// TwinCAT 3 PLC project HardwareSimulator
// ProgramVersion: 3.1.4024.0
// libraries:
//   Tc2_Standard, * (Beckhoff Automation GmbH)
//   Tc2_System, * (Beckhoff Automation GmbH)
//   Tc2_Utilities, * (Beckhoff Automation GmbH)
//   Tc3_Module, * (Beckhoff Automation GmbH)
//   VisuSymbols,3.5.10.0,System
// project tree:
//   / GlobalTextList.TcGTLO (not stored), PlcTask.TcTTO (not stored), Visualization Manager.TcVMO (not stored)
//   POUs/ MAIN.TcPOU, SIM_ValveWithFB.TcPOU, SIM_ValveWithDoubleFB.TcPOU, SIM_MOVITRAC_B.TcPOU (not stored)
//   VISUs/ Visualization.TcVIS (not stored)
// (motion and I/O tree: see PLC project cleanroomconnect)
// real-time tasks:
//   TASK PlcTask: cycle T#10ms, priority 20, ADS port 350
//   TASK PlcTask1: cycle T#10ms, priority 21, ADS port 351
//   TASK VISU_TASK: cycle T#200000us, priority 30, ADS port 352
// variable links:
//   CleanroomConnect/CleanroomConnect Instance <-> HardwareSimulator/HardwareSimulator Instance
//     PlcTask Inputs/GVL_Modules.g_emDockingInterface.s_cmDockingClampsLower.I_bStaValveIsOff <-> PlcTask Outputs/MAIN.simDockingClampLower.Q_bStaFeedbackOff
//     PlcTask Inputs/GVL_Modules.g_emDockingInterface.s_cmDockingClampsLower.I_bStaValveIsOff2 <-> PlcTask Outputs/MAIN.simDockingClampLower.Q_bStaFeedbackOff2
//     PlcTask Inputs/GVL_Modules.g_emDockingInterface.s_cmDockingClampsLower.I_bStaValveIsOn <-> PlcTask Outputs/MAIN.simDockingClampLower.Q_bStaFeedbackOn
//     PlcTask Inputs/GVL_Modules.g_emDockingInterface.s_cmDockingClampsLower.I_bStaValveIsOn2 <-> PlcTask Outputs/MAIN.simDockingClampLower.Q_bStaFeedbackOn2
//     PlcTask Inputs/GVL_Modules.g_emDockingInterface.s_cmDockingClampsUpper.I_bStaValveIsOff <-> PlcTask Outputs/MAIN.simDockingClampUpper.Q_bStaFeedbackOff
//     PlcTask Inputs/GVL_Modules.g_emDockingInterface.s_cmDockingClampsUpper.I_bStaValveIsOff2 <-> PlcTask Outputs/MAIN.simDockingClampUpper.Q_bStaFeedbackOff2
//     PlcTask Inputs/GVL_Modules.g_emDockingInterface.s_cmDockingClampsUpper.I_bStaValveIsOn <-> PlcTask Outputs/MAIN.simDockingClampUpper.Q_bStaFeedbackOn
//     PlcTask Inputs/GVL_Modules.g_emDockingInterface.s_cmDockingClampsUpper.I_bStaValveIsOn2 <-> PlcTask Outputs/MAIN.simDockingClampUpper.Q_bStaFeedbackOn2
//     PlcTask Inputs/GVL_Modules.g_emDockingInterface.s_cmDoorOpener.I_bStaValveIsOff <-> PlcTask Outputs/MAIN.simDoorOpener.Q_bStaFeedbackOff
//     PlcTask Inputs/GVL_Modules.g_emDockingInterface.s_cmDoorOpener.I_bStaValveIsOn <-> PlcTask Outputs/MAIN.simDoorOpener.Q_bStaFeedbackOn
//     PlcTask Inputs/GVL_Modules.g_emDockingInterface.s_cmDoorShutter.I_bStaValveIsOff <-> PlcTask Outputs/MAIN.simDoorShutter.Q_bStaFeedbackOff
//     PlcTask Inputs/GVL_Modules.g_emDockingInterface.s_cmDoorShutter.I_bStaValveIsOn <-> PlcTask Outputs/MAIN.simDoorShutter.Q_bStaFeedbackOn
//     PlcTask Inputs/GVL_Modules.g_emDockingInterface.s_cmUnlockingPinLower.I_bStaValveIsOff <-> PlcTask Outputs/MAIN.simUnlockPinLower.Q_bStaFeedbackOff
//     PlcTask Inputs/GVL_Modules.g_emDockingInterface.s_cmUnlockingPinLower.I_bStaValveIsOn <-> PlcTask Outputs/MAIN.simUnlockPinLower.Q_bStaFeedbackOn
//     PlcTask Inputs/GVL_Modules.g_emDockingInterface.s_cmUnlockingPinUpper.I_bStaValveIsOff <-> PlcTask Outputs/MAIN.simUnlockPinUpper.Q_bStaFeedbackOff
//     PlcTask Inputs/GVL_Modules.g_emDockingInterface.s_cmUnlockingPinUpper.I_bStaValveIsOn <-> PlcTask Outputs/MAIN.simUnlockPinUpper.Q_bStaFeedbackOn
//     PlcTask Inputs/GVL_Modules.g_emPalletConveyor.s_cmCentringUnit.I_bStaValveIsOff <-> PlcTask Outputs/MAIN.simCentring.Q_bStaFeedbackOff
//     PlcTask Inputs/GVL_Modules.g_emPalletConveyor.s_cmCentringUnit.I_bStaValveIsOff2 <-> PlcTask Outputs/MAIN.simCentring.Q_bStaFeedbackOff2
//     PlcTask Inputs/GVL_Modules.g_emPalletConveyor.s_cmCentringUnit.I_bStaValveIsOn <-> PlcTask Outputs/MAIN.simCentring.Q_bStaFeedbackOn
//     PlcTask Inputs/GVL_Modules.g_emPalletConveyor.s_cmCentringUnit.I_bStaValveIsOn2 <-> PlcTask Outputs/MAIN.simCentring.Q_bStaFeedbackOn2
//     PlcTask Inputs/GVL_Modules.g_emPalletConveyor.s_cmPalletConveyor.I_bStaMotorIsRunning <-> PlcTask Outputs/MAIN.sim_MOVITRAC_B.Q_bStaMotorIsRunning
//     PlcTask Inputs/GVL_Modules.g_emPalletConveyor.s_cmPalletConveyor.I_bStaReadyForOperation <-> PlcTask Outputs/MAIN.sim_MOVITRAC_B.Q_bStaReadyForOperation
//     PlcTask Outputs/GVL_Modules.g_emDockingInterface.s_cmDockingClampsLower.Q_bCmdOff <-> PlcTask Inputs/MAIN.simDockingClampLower.I_bCmdValveOff
//     PlcTask Outputs/GVL_Modules.g_emDockingInterface.s_cmDockingClampsLower.Q_bCmdOn <-> PlcTask Inputs/MAIN.simDockingClampLower.I_bCmdValveOn
//     PlcTask Outputs/GVL_Modules.g_emDockingInterface.s_cmDockingClampsUpper.Q_bCmdOff <-> PlcTask Inputs/MAIN.simDockingClampUpper.I_bCmdValveOff
//     PlcTask Outputs/GVL_Modules.g_emDockingInterface.s_cmDockingClampsUpper.Q_bCmdOn <-> PlcTask Inputs/MAIN.simDockingClampUpper.I_bCmdValveOn
//     PlcTask Outputs/GVL_Modules.g_emDockingInterface.s_cmDoorOpener.Q_bCmdOff <-> PlcTask Inputs/MAIN.simDoorOpener.I_bCmdValveOff
//     PlcTask Outputs/GVL_Modules.g_emDockingInterface.s_cmDoorOpener.Q_bCmdOn <-> PlcTask Inputs/MAIN.simDoorOpener.I_bCmdValveOn
//     PlcTask Outputs/GVL_Modules.g_emDockingInterface.s_cmDoorShutter.Q_bCmdOff <-> PlcTask Inputs/MAIN.simDoorShutter.I_bCmdValveOff
//     PlcTask Outputs/GVL_Modules.g_emDockingInterface.s_cmDoorShutter.Q_bCmdOn <-> PlcTask Inputs/MAIN.simDoorShutter.I_bCmdValveOn
//     PlcTask Outputs/GVL_Modules.g_emDockingInterface.s_cmUnlockingPinLower.Q_bCmdOff <-> PlcTask Inputs/MAIN.simUnlockPinLower.I_bCmdValveOff
//     PlcTask Outputs/GVL_Modules.g_emDockingInterface.s_cmUnlockingPinLower.Q_bCmdOn <-> PlcTask Inputs/MAIN.simUnlockPinLower.I_bCmdValveOn
//     PlcTask Outputs/GVL_Modules.g_emDockingInterface.s_cmUnlockingPinUpper.Q_bCmdOff <-> PlcTask Inputs/MAIN.simUnlockPinUpper.I_bCmdValveOff
//     PlcTask Outputs/GVL_Modules.g_emDockingInterface.s_cmUnlockingPinUpper.Q_bCmdOn <-> PlcTask Inputs/MAIN.simUnlockPinUpper.I_bCmdValveOn
//     PlcTask Outputs/GVL_Modules.g_emPalletConveyor.s_cmCentringUnit.Q_bCmdOff <-> PlcTask Inputs/MAIN.simCentring.I_bCmdValveOff
//     PlcTask Outputs/GVL_Modules.g_emPalletConveyor.s_cmCentringUnit.Q_bCmdOn <-> PlcTask Inputs/MAIN.simCentring.I_bCmdValveOn
//     PlcTask Outputs/GVL_Modules.g_emPalletConveyor.s_cmPalletConveyor.Q_bCmdEnable <-> PlcTask Inputs/MAIN.sim_MOVITRAC_B.I_bCmdEnable
//     PlcTask Outputs/GVL_Modules.g_emPalletConveyor.s_cmPalletConveyor.Q_bCmdReset <-> PlcTask Inputs/MAIN.sim_MOVITRAC_B.I_bCmdReset
//     PlcTask Outputs/GVL_Modules.g_emPalletConveyor.s_cmPalletConveyor.Q_bCmdStartCCW <-> PlcTask Inputs/MAIN.sim_MOVITRAC_B.I_bCmdStartCCW
//     PlcTask Outputs/GVL_Modules.g_emPalletConveyor.s_cmPalletConveyor.Q_bCmdStartCW <-> PlcTask Inputs/MAIN.sim_MOVITRAC_B.I_bCmdStartCW

// ---- POUs/MAIN.TcPOU
PROGRAM MAIN
VAR
	//EM Pallet Transport
	sim_MOVITRAC_B : SIM_MOVITRAC_B;
	simCentring : SIM_ValveWithDoubleFB;	

	//EM Docking Interface
	simDockingClampUpper : SIM_ValveWithDoubleFB;
	simDockingClampLower : SIM_ValveWithDoubleFB;
	simUnlockPinUpper : SIM_ValveWithFB;
	simUnlockPinLower : SIM_ValveWithFB;
	simDoorOpener : SIM_ValveWithFB;
	simDoorShutter : SIM_ValveWithFB;
	simDoorOpenerAlmostClosed AT %Q* : BOOL;
	tonDoorOpenerAlmosClosed : TON;
END_VAR


//EM Pallet Conveyor
sim_MOVITRAC_B();
simCentring();

//EM Docking Interface
simDockingClampUpper();
simDockingClampLower();
simUnlockPinUpper();
simUnlockPinLower();
simDoorOpener();
simDoorShutter();

tonDoorOpenerAlmosClosed(IN := simDoorOpener.q_bStaValveOff, PT := T#1S);
simDoorOpenerAlmostClosed := tonDoorOpenerAlmosClosed.Q;

END_PROGRAM

// ---- POUs/SIM_ValveWithDoubleFB.TcPOU
FUNCTION_BLOCK SIM_ValveWithDoubleFB
VAR 
	// Outputs from PLC --> HW
	I_bCmdValveOn AT %I* : BOOL;
	I_bCmdValveOff AT %I* : BOOL;
	
	// Inputs from HW --> PLC
	Q_bStaFeedbackOn AT %Q* : BOOL;
	Q_bStaFeedbackOff AT %Q* : BOOL;
	Q_bStaFeedbackOn2 AT %Q* : BOOL;
	Q_bStaFeedbackOff2 AT %Q* : BOOL;
	
	s_tonOn : TON;
	s_tonOff : TON;
	
END_VAR

VAR_OUTPUT
	q_bStaValveOn : BOOL;
	q_bStaValveOff : BOOL;
END_VAR


s_tonOn(IN := I_bCmdValveOn AND NOT(I_bCmdValveOff), PT := T#2S);

IF s_tonOn.Q THEN
	Q_bStaFeedbackOn := TRUE;
	Q_bStaFeedbackOn2 := TRUE;
ELSIF I_bCmdValveOff THEN
	Q_bStaFeedbackOn := FALSE;
	Q_bStaFeedbackOn2 := FALSE;
END_IF	
	
s_tonOff(IN := I_bCmdValveOff AND NOT(I_bCmdValveOn), PT := T#2S);

IF s_tonOff.Q THEN
	Q_bStaFeedbackOff := TRUE;
	Q_bStaFeedbackOff2 := TRUE;
ELSIF I_bCmdValveOn THEN
	Q_bStaFeedbackOff := FALSE;
	Q_bStaFeedbackOff2 := FALSE;
END_IF

q_bStaValveOn := I_bCmdValveOn;
q_bStaValveOff := I_bCmdValveOff;

END_FUNCTION_BLOCK

// ---- POUs/SIM_ValveWithFB.TcPOU
FUNCTION_BLOCK SIM_ValveWithFB
VAR 
	// Outputs from PLC --> HW
	I_bCmdValveOn AT %I* : BOOL;
	I_bCmdValveOff AT %I* : BOOL;
	
	// Inputs from HW --> PLC
	Q_bStaFeedbackOn AT %Q* : BOOL;
	Q_bStaFeedbackOff AT %Q* : BOOL;
	
	s_tonOn : TON;
	s_tonOff : TON;
	
END_VAR

VAR_OUTPUT
	q_bStaValveOn : BOOL;
	q_bStaValveOff : BOOL;
END_VAR

s_tonOn(IN := I_bCmdValveOn AND NOT(I_bCmdValveOff), PT := T#2S);

IF s_tonOn.Q THEN
	Q_bStaFeedbackOn := TRUE;
ELSIF I_bCmdValveOff THEN
	Q_bStaFeedbackOn := FALSE;
END_IF	
	
s_tonOff(IN := I_bCmdValveOff AND NOT(I_bCmdValveOn), PT := T#2S);

IF s_tonOff.Q THEN
	Q_bStaFeedbackOff := TRUE;
ELSIF I_bCmdValveOn THEN
	Q_bStaFeedbackOff := FALSE;
END_IF

q_bStaValveOn := I_bCmdValveOn;
q_bStaValveOff := I_bCmdValveOff;

END_FUNCTION_BLOCK
